// TIA Portal V21 export
VAR_GLOBAL   // PLC tag table "KAllRicetta"
END_VAR
VAR_GLOBAL CONSTANT   // user constants
   KAllRicetta_IncoerenzaAltezzaCubo : Int := 1;
   KAllRicetta_QuoteFuoriRange : Int := 2;
END_VAR
